// TIA Portal V20 export
DATA_BLOCK "Simulation"   // DB134
TITLE = Simulation
// Simulation data
// stored: MemoryReserve 100
   VAR
      data : "LAF_typeSimulation";
   END_VAR
BEGIN
   data.simulationActiveHmi := true;
END_DATA_BLOCK
